(* CODESYS project e!C_AT_CMD_SMS_Test_1.ecp

Project tree, tasks and I/O mapping:
  Controller : 750-8202 PFC200 2ETH RS, WAGO, order no. 0750-8202, version 5.11.1.16
    application Application
      libraries: ; WagoAppSocket, * (WAGO); WagoAppSerial_Sms, * (WAGO)
      task PLC_Task (cyclic, interval t#10ms, priority 15) calls PLC_PRG
      program PLC_PRG [ST]
      data type DUT_StringAndBytes
      global variables GCL_SMS
      data type DUT_SmsExchangeType
      function block fbModemSms [ST]: AT_CMD_SMS_CONSTRUCT, AT_CMD_SMS_EVALUATE, AT_CMD_SMS_SEQUENCER
    DeviceAdapter
    Kbus : Kbus, WAGO, version 1.4.0.2
        unmapped channels: K-BUS diagnostics
    MODBUS
      MODBUS : MODBUS, WAGO, order no. n/a, version 1.1.1.15
    Serial
      COM1 : COM1, WAGO, version 0.0.0.19
*)

// Controller/Application/DUT_StringAndBytes
TYPE DUT_StringAndBytes :
UNION
	abBuffer: ARRAY[1..GCL_SMS.LIM_OF_SMS_LENGTH] OF BYTE;
	sBuffer: STRING(GCL_SMS.LIM_OF_SMS_LENGTH);
END_UNION
END_TYPE

// Controller/Application/DUT_SmsExchangeType
{attribute 'qualified_only'}
{attribute 'strict'}
TYPE DUT_SmsExchangeType :
(
	eSmsExchangeSend := 1,
	eSmsExchangeRead := 2,
	eSmsExchangeDelete := 3
);
END_TYPE

// Controller/Application/GCL_SMS
{attribute 'qualified_only'}
VAR_GLOBAL CONSTANT
	LIM_OF_SMS_DESTINATIONS: INT := 5;
	LIM_OF_SMS_LENGTH: INT := 1000;	
END_VAR

// Controller/Application/PLC_PRG
PROGRAM PLC_PRG
VAR
	fbModemSms_Test: fbModemSms;
	sModemIp: STRING := '192.168.1.1';
	eSmsExchangeType: DUT_SmsExchangeType := DUT_SmsExchangeType.eSmsExchangeSend;
	xSmsExchangeStart: BOOL;
	sSmsReadMessage: STRING(GCL_SMS.LIM_OF_SMS_LENGTH);
	sSmsSendMessage: STRING(GCL_SMS.LIM_OF_SMS_LENGTH) := 'SMS New Test...';
	asSmsDestination: ARRAY[1..GCL_SMS.LIM_OF_SMS_DESTINATIONS] OF STRING := [GCL_SMS.LIM_OF_SMS_DESTINATIONS('+4797195836')];
	xSmsSend: BOOL;
	R_TRIG_SmsSend: R_TRIG;
END_VAR



fbModemSms_Test(
	sModemIp			:= sModemIp, 
	eSmsExchangeType	:= eSmsExchangeType, 
	asSmsDestination	:= asSmsDestination, 
	sSmsSendMessage		:= sSmsSendMessage, 
	sSmsReadMessage		:= sSmsReadMessage,
	xSmsExchangeStart	:= xSmsExchangeStart);

IF (xSmsExchangeStart = FALSE) THEN
	R_TRIG_SmsSend(CLK:= xSmsSend, Q=>xSmsExchangeStart);
END_IF

END_PROGRAM

// Controller/Application/fbModemSms
FUNCTION_BLOCK fbModemSms
VAR_INPUT
	sModemIp: STRING := '192.168.1.1'; (* IP address of Maestro modem *)
	eSmsExchangeType: DUT_SmsExchangeType := DUT_SmsExchangeType.eSmsExchangeSend;
	asSmsDestination: ARRAY[1..GCL_SMS.LIM_OF_SMS_DESTINATIONS] OF STRING := [GCL_SMS.LIM_OF_SMS_DESTINATIONS('+4797195836')];
	sSmsSendMessage: STRING(GCL_SMS.LIM_OF_SMS_LENGTH) := 'Test SMS...';
END_VAR
VAR_IN_OUT
	sSmsReadMessage: STRING(GCL_SMS.LIM_OF_SMS_LENGTH);
	xSmsExchangeStart: BOOL;
END_VAR
VAR_OUTPUT
END_VAR
VAR
	DUT_AT_CMD_SMS_TX: DUT_StringAndBytes;
	DUT_AT_CMD_SMS_RX: DUT_StringAndBytes;
	iSmsDestinationIndex: INT;
	iAtCmdSmsState: INT;
	FbTcpClient_AT_CMD_SMS: WagoAppSocket.FbTcpClient;
	wPort: WORD := 5555;
	oStatus: FbResult;
	xOpen: BOOL:= TRUE;
	xIsOpen: BOOL;
	xIsIdle: BOOL;
	xError: BOOL;
	xTxTrigger: BOOL;
	udiTxNBytes: UDINT;
	udiRxIndex: UDINT;
	xRxBufferFull: BOOL;
	xRxOverflow: BOOL;
	xResetStatus: BOOL;
	xKeepAlive_Enable: BOOL := FALSE;
	tKeepAlive_MaxIdleTime: TIME := T#10S;
	tKeepAlive_Interval: TIME := T#1S;
	udiKeepAlive_Probes: UDINT := 5;
	TON_ModemMonitor: TON;
	tModemTimeout: TIME := T#2s;
END_VAR

FbTcpClient_AT_CMD_SMS(
	oStatus					=> oStatus, 
	xOpen					:= xOpen, 
	xIsOpen					=> xIsOpen, 
	xIsIdle					=> xIsIdle, 
	xError					=> xError, 
	xTxTrigger				:= xTxTrigger, 
	pTxBuffer				:= ADR(DUT_AT_CMD_SMS_TX.abBuffer), 
	udiTxNBytes				:= LEN(DUT_AT_CMD_SMS_TX.sBuffer)+1, 
	pRxBuffer				:= ADR(DUT_AT_CMD_SMS_RX.abBuffer), 
	udiRxBufferSize			:= SIZEOF(DUT_AT_CMD_SMS_RX.abBuffer), 
	udiRxIndex				:= udiRxIndex, 
	xRxBufferFull			=> xRxBufferFull, 
	xRxOverflow				=> xRxOverflow, 
	xResetStatus			:= xResetStatus, 
	sServerName				:= sModemIp, 
	wPort					:= wPort, 
	xKeepAlive_Enable		:= xKeepAlive_Enable, 
	tKeepAlive_MaxIdleTime	:= tKeepAlive_MaxIdleTime, 
	tKeepAlive_Interval		:= tKeepAlive_Interval, 
	udiKeepAlive_Probes		:= udiKeepAlive_Probes);

AT_CMD_SMS_SEQUENCER();

ACTION AT_CMD_SMS_CONSTRUCT:

IF (eSmsExchangeType = DUT_SmsExchangeType.eSmsExchangeSend) THEN (* SMS Send *)
	DUT_AT_CMD_SMS_TX.sBuffer := 'AT#SENDSMS=';
	DUT_AT_CMD_SMS_TX.sBuffer := CONCAT(DUT_AT_CMD_SMS_TX.sBuffer, '"');
	DUT_AT_CMD_SMS_TX.sBuffer := CONCAT(DUT_AT_CMD_SMS_TX.sBuffer, asSmsDestination[iSmsDestinationIndex]);
	DUT_AT_CMD_SMS_TX.sBuffer := CONCAT(DUT_AT_CMD_SMS_TX.sBuffer, '"');
	DUT_AT_CMD_SMS_TX.sBuffer := CONCAT(DUT_AT_CMD_SMS_TX.sBuffer, sSmsSendMessage);
	DUT_AT_CMD_SMS_TX.sBuffer := CONCAT(DUT_AT_CMD_SMS_TX.sBuffer, '$04');
ELSIF (eSmsExchangeType = DUT_SmsExchangeType.eSmsExchangeRead) THEN (* SMS Read *)
	DUT_AT_CMD_SMS_TX.sBuffer := 'AT#READSMS="ALL"$04';
ELSIF (eSmsExchangeType = DUT_SmsExchangeType.eSmsExchangeDelete) THEN (* SMS Delete *)
	DUT_AT_CMD_SMS_TX.sBuffer := 'AT#DELSMS="ALL"$04';
END_IF
DUT_AT_CMD_SMS_RX.sBuffer := '';
END_ACTION

ACTION AT_CMD_SMS_EVALUATE:


IF (eSmsExchangeType = DUT_SmsExchangeType.eSmsExchangeSend) THEN (* SMS Send *)
	IF (DUT_AT_CMD_SMS_RX.sBuffer = '') THEN
		(* TO DO: Evaluate Response After Sending SMS... *);
	END_IF
ELSIF (eSmsExchangeType = DUT_SmsExchangeType.eSmsExchangeRead) THEN (* SMS Read *)
	sSmsReadMessage := DUT_AT_CMD_SMS_RX.sBuffer;
ELSIF (eSmsExchangeType = DUT_SmsExchangeType.eSmsExchangeDelete) THEN (* SMS Delete *)
	IF (DUT_AT_CMD_SMS_RX.sBuffer = '') THEN
		(* TO DO: Evaluate Response After Deleting SMS... *);
	END_IF
END_IF
END_ACTION

ACTION AT_CMD_SMS_SEQUENCER:

CASE iAtCmdSmsState OF

	0:
		iSmsDestinationIndex := 1;
		iAtCmdSmsState := 1;
	1:
		IF (xSmsExchangeStart = TRUE) THEN
			iAtCmdSmsState := 2;
		END_IF
	2:
		xOpen := TRUE;
		IF (xIsOpen = TRUE) THEN
			TON_ModemMonitor(IN:= FALSE);
			iAtCmdSmsState := 10;
		ELSE
			TON_ModemMonitor(IN:= TRUE, PT:= tModemTimeout);
			IF (TON_ModemMonitor.Q = TRUE) THEN
				TON_ModemMonitor(IN:= FALSE);
				iAtCmdSmsState := 100;
			END_IF
		END_IF

	10:
		AT_CMD_SMS_CONSTRUCT();
		xTxTrigger := TRUE;
		udiRxIndex := 0;
		iAtCmdSmsState := 11;
	11:
		IF (xTxTrigger = FALSE) THEN
			AT_CMD_SMS_EVALUATE();
			xOpen := FALSE;
			IF (xIsOpen = FALSE) THEN
				iSmsDestinationIndex := iSmsDestinationIndex + 1;
				IF (iSmsDestinationIndex > GCL_SMS.LIM_OF_SMS_DESTINATIONS) THEN
					xSmsExchangeStart := FALSE;
					iSmsDestinationIndex := 1;
					iAtCmdSmsState := 1;
				ELSIF (asSmsDestination[iSmsDestinationIndex] = '') THEN
					xSmsExchangeStart := FALSE;
					iSmsDestinationIndex := 1;
					iAtCmdSmsState := 1;
				ELSE
					iAtCmdSmsState := 2;
				END_IF
			END_IF
		END_IF

	100:(* Modem connection error *)
		xOpen := FALSE;
		xTxTrigger := FALSE;
		IF (xIsOpen = FALSE) THEN
			iAtCmdSmsState := 1;
		END_IF

END_CASE
END_ACTION

END_FUNCTION_BLOCK
